{attribute 'qualified_only'}
VAR_GLOBAL
	Charger		: ARRAY[1..8] OF ST_Echo_MCP;
	GLSLoad		: ST_ChargeTime;
	Section : ARRAY[1..4] OF ST_Echo_Section;
END_VAR

(* stored: Version 1.1.0.1, ProductVersion 3.1.4024.11
   GVL TxMainPLC: Id {af7db7f0-277a-4aaa-8bec-b684ccb4316c} *)
